FUNCTION_BLOCK FB_OpenFile

VAR
	fbStartProcess : NT_StartProcess := (NETID := '',TMOUT := T#5S );
	bError : BOOL;
END_VAR

fbStartProcess(PATHSTR := 'C:\Windows\notepad.exe',
				DIRNAME := 'D:\Temp\',
				COMNDLINE := 'Event.txt',
				START := TRUE
				);
bError := fbStartProcess.ERR;

END_FUNCTION_BLOCK

(* stored: Version 1.1.0.1, ProductVersion 3.1.4024.16
   POU FB_OpenFile: Id {1cf29e12-b6d9-442c-996b-692ed06927eb}, SpecialFunc None *)
